// TIA Portal V17 export
// export: Created 2026-04-13T11:12:41.7704649Z, ExportSetting WithDefaults, DisplayName Totally Integrated Automation Portal, DisplayVersion V17 Update 4, DisplayName TIA Portal Openness, DisplayVersion V17 Update 4, DisplayName TIA Portal Version Control Interface, DisplayVersion V17, DisplayName SINAMICS Startdrive Advanced, DisplayVersion V17, DisplayName SINAMICS Startdrive G130, G150, S120, S150, SINAMICS MV, S210, DisplayVersion V17, DisplayName SINAMICS Startdrive G110M, G120, G120C, G120D, G120P, G115D, DisplayVersion V17, DisplayName STEP 7 Professional, DisplayVersion V17 Update 4, DisplayName STEP 7 Safety, DisplayVersion V17, DisplayName WinCC Professional, DisplayVersion V17 Update 4
FUNCTION_BLOCK "B2_循环下料控制_F"   // FB38, SCL
{ S7_Optimized_Access := 'TRUE' }
VERSION : 0.1
// stored: AutoNumber true, IsIECCheckEnabled false, IsRetainMemResEnabled false, MemoryReserve 100, SetENOAutomatically false, UDAEnableTagReadback false
   VAR_INPUT
      启动按钮 : Bool;   // 启动循环下料的按钮
      停止按钮 : Bool;   // 停止循环下料的按钮
      SF上阀打开时间 : Real := 10.0;
      SF上阀关闭时间 : Real := 5.0;
      XF下阀打开时间 : Real := 10.0;
      XF下阀关闭时间 : Real := 5.0;
   END_VAR
   VAR_OUTPUT
      上阀控制 : Bool;   // 上阀控制信号 TRUE=打开
      下阀控制 : Bool;   // 下阀控制信号 TRUE=打开
      当前状态 : Int;   // 当前状态显示
      运行状态 : Bool;   // 系统运行状态
   END_VAR
   VAR
      状态 : Int := 0;   // 状态机变量：0=停止，1=上阀打开，2=上阀关闭，3=下阀打开，4=下阀关闭
      计时器 { S7_SetPoint := 'True'} : TON_TIME;   // 计时器
      上次状态 : Int := 0;   // 记录上一个状态
      启动边沿检测 { S7_SetPoint := 'True'} : R_TRIG;   // 启动按钮上升沿检测
      停止边沿检测 { S7_SetPoint := 'True'} : R_TRIG;   // 停止按钮上升沿检测
      上阀打开时间 : Time;   // 上阀打开持续时间 默认10秒
      上阀关闭时间 : Time;   // 上阀关闭持续时间 默认5秒
      下阀打开时间 : Time;   // 下阀打开持续时间 默认10秒
      下阀关闭时间 : Time;   // 下阀关闭持续时间 默认5秒
   END_VAR
BEGIN
       // 检测启动按钮上升沿
       // REAL_MS_TO_TIME := DINT_TO_TIME(REAL_TO_DINT(IN_REAL * 1000.0));
       // REAL_MS_TO_TIME := DINT_TO_TIME(REAL_TO_DINT(IN_REAL));
       #上阀打开时间 := DINT_TO_TIME(REAL_TO_DINT(#SF上阀打开时间 * 1000.0));
       #上阀关闭时间 := DINT_TO_TIME(REAL_TO_DINT(#SF上阀关闭时间 * 1000.0));
       #下阀打开时间 := DINT_TO_TIME(REAL_TO_DINT(#XF下阀打开时间 * 1000.0));
       #下阀关闭时间 := DINT_TO_TIME(REAL_TO_DINT(#XF下阀关闭时间 * 1000.0));

      // TotalMS := TIME_TO_DINT(IN_TIME); // 转换为毫秒
       // TIME_TO_REAL_MS := DINT_TO_REAL(TIME_TO_DINT(IN_TIME));
       // TIME_TO_REAL_S := DINT_TO_REAL(TIME_TO_DINT(IN_TIME)) / 1000.0;
       #启动边沿检测(CLK := #启动按钮);

       // 检测停止按钮上升沿
       #停止边沿检测(CLK := #停止按钮);

       // 处理启动/停止
       IF #停止边沿检测.Q THEN
           #状态 := 0;  // 停止
           #运行状态 := FALSE;
       ELSIF #启动边沿检测.Q AND #状态 = 0 THEN
           #状态 := 1;  // 启动，从上阀打开开始
           #运行状态 := TRUE;
       END_IF;

       // 状态机逻辑
       CASE #状态 OF
           0:  // 停止状态
               #上阀控制 := FALSE;
               #下阀控制 := FALSE;
               #计时器(IN := FALSE,
                    PT := T#0S);

           1:  // 状态1：上阀打开
               #上阀控制 := TRUE;
               #下阀控制 := FALSE;

               // 如果状态刚刚变化，重置计时器
               IF #上次状态 <> #状态 THEN
                   #计时器(IN := FALSE,
                        PT := #上阀打开时间);
                   #上次状态 := #状态;
               END_IF;

               // 启动计时器
               #计时器(IN := TRUE,
                    PT := #上阀打开时间);

               // 当计时器到达设定时间，切换到下一个状态
               IF #计时器.Q THEN
                   #状态 := 2;  // 切换到上阀关闭状态
               END_IF;

           2:  // 状态2：上阀关闭
               #上阀控制 := FALSE;
               #下阀控制 := FALSE;

               // 如果状态刚刚变化，重置计时器
               IF #上次状态 <> #状态 THEN
                   #计时器(IN := FALSE,
                        PT := #上阀关闭时间);
                   #上次状态 := #状态;
               END_IF;

               // 启动计时器
               #计时器(IN := TRUE,
                    PT := #上阀关闭时间);

               // 当计时器到达设定时间，切换到下一个状态
               IF #计时器.Q THEN
                   #状态 := 3;  // 切换到下阀打开状态
               END_IF;

           3:  // 状态3：下阀打开
               #上阀控制 := FALSE;
               #下阀控制 := TRUE;

               // 如果状态刚刚变化，重置计时器
               IF #上次状态 <> #状态 THEN
                   #计时器(IN := FALSE,
                        PT := #下阀打开时间);
                   #上次状态 := #状态;
               END_IF;

               // 启动计时器
               #计时器(IN := TRUE,
                    PT := #下阀打开时间);

               // 当计时器到达设定时间，切换到下一个状态
               IF #计时器.Q THEN
                   #状态 := 4;  // 切换到下阀关闭状态
               END_IF;

           4:  // 状态4：下阀关闭
               #上阀控制 := FALSE;
               #下阀控制 := FALSE;

               // 如果状态刚刚变化，重置计时器
               IF #上次状态 <> #状态 THEN
                   #计时器(IN := FALSE,
                        PT := #下阀关闭时间);
                   #上次状态 := #状态;
               END_IF;

               // 启动计时器
               #计时器(IN := TRUE,
                    PT := #下阀关闭时间);

               // 当计时器到达设定时间，切换回第一个状态
               IF #计时器.Q THEN
                   #状态 := 1;  // 返回上阀打开状态，完成一个循环
               END_IF;

           ELSE  // 异常状态处理
               #状态 := 0;  // 恢复到停止状态
               #上阀控制 := FALSE;
               #下阀控制 := FALSE;
       END_CASE;

       // 更新输出状态
       #当前状态 := #状态;
END_FUNCTION_BLOCK
